{attribute 'pack_mode' := '1'}
TYPE TRunDataReject :
STRUCT
	eRejectStatus		: TRejectStatus;
END_STRUCT
END_TYPE

(* stored: Version 1.1.0.1, ProductVersion 3.1.4022.12
   DUT TRunDataReject: Id {938f095a-3981-45e1-9176-758865eaa9c5} *)
